FUNCTION_BLOCK FB_ContainerDefGrid EXTENDS FB_ContainerBase
VAR_INPUT
END_VAR
VAR_OUTPUT
END_VAR
VAR
  fBImageDeformation : FB_ImageDeformation;  
END_VAR

fBImageDeformation();                       // call run cyclic image deformation
fBImageDeformation.LogLevel := LogLevel;    // distribute container logLevel to image deformation fb

METHOD AbortDeformation : BOOL
VAR_INPUT
  sReason : STRING;
  Src     : REFERENCE TO T_ErrSrc;
END_VAR
LogWarning(F_Concat2('Abort deformation: ', sReason));  // log reason
setError(ErrDef:=EC_DefGrid.ecDefGrid_DefGridAbort, Src:=Src); // tag ct as error
fBImageDeformation.abort();  // abort deformation
END_METHOD

METHOD AddCamPoint : BOOL
VAR_INPUT
  sPoint : ST_DeformationPointAccurate;
END_VAR
AddCamPoint := fBImageDeformation.addCamPoint(sNewPoint:=sPoint);
END_METHOD

(*
  Create a container, build very basics.
*)
METHOD Create : BOOL
VAR_INPUT
	nCTId	            : DINT;     (* a container identifier *)
	nCTIndex	        : UDINT;	  (* memory index (array index if CT in CT array) *)
END_VAR
SUPER^.Create(nCTId:=nCTId, nCTIndex:=nCTIndex);
fBImageDeformation.reset();
fBImageDeformation.nProcessId := THIS^.pCT^.iId;
END_METHOD

(*
  Shift in x [SubPx]
*)
PROPERTY fDxShift : LREAL
GET
VAR
  errCtr : UDINT;
END_VAR
fDxShift := fBImageDeformation._nDxShift;
END_GET
END_PROPERTY

(*
  Shift in y [Px]
*)
PROPERTY fDyShift : LREAL
GET
VAR
  errCtr : UDINT;
END_VAR
fDyShift := fBImageDeformation._nDyShift;
END_GET
END_PROPERTY

(*
  get a deformation point.
  :returns: TRUE if successful
*)
METHOD getDeformationPoint : BOOL;
VAR_INPUT
  nCol : UDINT;   // col select
  nRow : UDINT;   // row select
END_VAR
VAR_OUTPUT
  sPoint : ST_DeformationPointAccurate;
END_VAR
getDeformationPoint := fBImageDeformation.getDeformationPoint(nCol:=nCol, nRow:=nRow, sPoint=>sPoint);
END_METHOD

(*
  Deformation state of CT.
  :return:  TRUE in case of error -> any deformation error
*)
METHOD getDeformationStatus : BOOL
VAR_INPUT
END_VAR
VAR_OUTPUT
  eDStep: E_DeformationStep;// deformation step
  bDone : BOOL;             // deformation done
  bBusy : BOOL;             // deformation is busy
  nErrorId : UDINT;         // error id in case of error
  tExecutionTime : TIME;    // script update execution time?
END_VAR
getDeformationStatus := fBImageDeformation.bError;

eDStep:= fBImageDeformation.eStep;
bBusy := fBImageDeformation.bBusy;
bDone := fBImageDeformation.bDone;
nErrorId := fBImageDeformation.nErrorId;
tExecutionTime := fBImageDeformation.tExecutionTime;
END_METHOD

PROPERTY nAvailableGridCols : UDINT
GET
nAvailableGridCols := fBImageDeformation._nGridCols;
END_GET
END_PROPERTY

PROPERTY nAvailableGridPoints : UDINT
GET
nAvailableGridPoints := fBImageDeformation.nAvailableGridPoints;
END_GET
END_PROPERTY

PROPERTY PUBLIC nRegisteredCameraPoints : UDINT
GET
nRegisteredCameraPoints := fBImageDeformation._nCamPoints;
END_GET
END_PROPERTY

PROPERTY sDefGridSettings : ST_DefGridSettings
GET
sDefGridSettings := fBImageDeformation.sDefGridSettings;
END_GET
SET
fBImageDeformation.sDefGridSettings := sDefGridSettings;
END_SET
END_PROPERTY

METHOD SetupDeformation
VAR_INPUT
  eCameraMode : E_CameraMode;
END_VAR
// update mode
fBImageDeformation.eMode := eCameraMode;
END_METHOD

METHOD StartDeformation
VAR_INPUT
  eDeformationStep : E_DeformationStep;
  //nParam1 : UDINT;
END_VAR
IF eDeformationStep = E_DeformationStep.nothing THEN
  ; // do nothing
ELSIF eDeformationStep = E_DeformationStep.createdScriptContainer THEN
  ;
ELSIF eDeformationStep = E_DeformationStep.cameraStarted THEN
  fBImageDeformation.startCamera(
    fStartDefPos:=DINT_TO_LREAL(THIS^.GetPos(nPosDomain:=E_PosDomain.pos_px))
  );
END_IF


// update step if it is bigger
IF fBImageDeformation.eStep < eDeformationStep THEN
  fBImageDeformation.eStep := eDeformationStep;
  LogLvl(Lvl:=E_LogSeverity.Debug, Msg:=F_Concat2('StartDeformation: step=', TO_STRING(eDeformationStep)));
END_IF
END_METHOD

(*
  Updates deformation module (max. in given interval)
*)
METHOD PUBLIC UpdateDeformation : BOOL
VAR_INPUT
  fUpdateInterval : LREAL;  // deformation module update interval [px]
END_VAR
fBImageDeformation.updateDeformation(
  fPos:=THIS^.GetPos(nPosDomain:=E_PosDomain.pos_px), 
  fUpdateInterval:=fUpdateInterval
);
END_METHOD

END_FUNCTION_BLOCK

(* stored: Version 1.1.0.1, ProductVersion 3.1.4024.3
   POU FB_ContainerDefGrid: Id {2d8beb5a-7741-4f53-9b5d-5bba1cb243c4}, SpecialFunc None
   Method AbortDeformation: Id {f4e769e7-fdcb-497a-869a-11c396829281}
   Method AddCamPoint: Id {c9a7845c-22a0-4577-acbe-8954df2e199f}
   Method Create: Id {e7db097f-b805-4a15-997e-aea4a4252e85}
   Property fDxShift: Id {f4b62b6e-2ae9-4fbc-b999-716d94294e90}
   Get Get: Id {66c9eb50-0679-4295-8ac5-c47a55b9a9c4}
   Property fDyShift: Id {a1bfccb0-2d05-4dbc-897b-c5caf07669b4}
   Get Get: Id {1d2c50e2-c63a-41c7-9fdd-72e3032bf798}
   Method getDeformationPoint: Id {2c7c8e7c-37b2-43e1-90a8-ea784d68621e}
   Method getDeformationStatus: Id {ad3cfac4-eda3-4d41-892b-ffdca204925e}
   Property nAvailableGridCols: Id {61be60fa-e3b9-4821-925e-23b920d7bfd3}
   Get Get: Id {8f97e19b-db85-4e14-95e2-7bc242c47118}
   Property nAvailableGridPoints: Id {d70e9fbe-44b3-4e41-aa7d-d45874a9762c}
   Get Get: Id {a3e9e991-2e2d-4b0b-9b38-b97f16ba20be}
   Property nRegisteredCameraPoints: Id {f813e15a-dac8-4907-83e3-431c7dfe5c84}
   Get Get: Id {e0059d97-ca3c-4ec0-8b56-5e7d4cb3596c}
   Property sDefGridSettings: Id {f9976eb4-29cd-4f5b-9829-bbe8c23a9ab1}
   Get Get: Id {bebda86e-82b9-4a1b-b7e5-739d4c134a65}
   Set Set: Id {f3c77bb0-91d2-48af-bba1-f099e412f5dd}
   Method SetupDeformation: Id {fa9cfc27-a9f9-4b08-a02d-72b82e2069db}
   Method StartDeformation: Id {197196c8-f164-46d2-868e-8fff7b370e59}
   Method UpdateDeformation: Id {cb380da5-bcaa-4509-a9f1-3ad6d51f2b1a} *)
